        (* Warnung Revisionsschalter Aus *)
        ayWarningReporter[2].proPrio := 1;
	    ayWarningReporter[2].proHandLokal :=    xVerdiRevisionSwitchOff; 
        ayWarningReporter[2].metReport(			xSetReportIn					:= xVerdiRevisionSwitchOff,
												iReportID						:= 2,
												enReportTypeIn					:= CtaAppReport.enReportType.Warning,  
												enReportAcknowledgeTypeIn   	:= CtaAppReport.enReportAcknowledgeType.Auto,
												tDelay							:= T#0S, 
												ITF_BMK_IN						:= THIS^,			              
												pstReportTextListIn				:= ADR(GlobalKonstant.stReportTextListWarning),
												stOptionalReportText		    := '',   
												iRetryTilReportLock 		    := 0, 
												xResetCount         		    := FALSE,  
												tReset						    := T#24H);     

        (* Warnung Hand Aus *)      
        ayWarningReporter[3].proPrio := 3;  
		ayWarningReporter[3].proHandLokal :=    xIsHandOff; 
        ayWarningReporter[3].metReport(			xSetReportIn					:= xIsHandOff,
												iReportID						:= 3,
												enReportTypeIn					:= CtaAppReport.enReportType.Warning,  
												enReportAcknowledgeTypeIn   	:= CtaAppReport.enReportAcknowledgeType.Auto,
												tDelay							:= T#0S, 
												ITF_BMK_IN						:= THIS^,			              
												pstReportTextListIn				:= ADR(GlobalKonstant.stReportTextListWarning),
												stOptionalReportText		    := '',   
												iRetryTilReportLock 		    := 0, 
												xResetCount         		    := FALSE,  
												tReset						    := T#24H);                                  
                                
        (* Warnung Hand Ein *)    
        ayWarningReporter[4].proPrio := 3; 
		ayWarningReporter[4].proHandLokal :=    xIsHandOn;
        ayWarningReporter[4].metReport(			xSetReportIn					:= xIsHandOn,
												iReportID						:= 4,
												enReportTypeIn					:= CtaAppReport.enReportType.Warning,  
												enReportAcknowledgeTypeIn   	:= CtaAppReport.enReportAcknowledgeType.Auto,
												tDelay							:= T#0S, 
												ITF_BMK_IN						:= THIS^,			              
												pstReportTextListIn				:= ADR(GlobalKonstant.stReportTextListWarning),
												stOptionalReportText		    := '',   
												iRetryTilReportLock 		    := 0, 
												xResetCount         		    := FALSE,  
												tReset						    := T#24H);   
 
        (* Warnung Handmodul Motor *)   
        ayWarningReporter[5].proPrio := 4;  
		ayWarningReporter[5].proHandLokal :=    xVerdichterHand;
        ayWarningReporter[5].metReport(			xSetReportIn					:= xVerdichterHand,
												iReportID						:= 5,
												enReportTypeIn					:= CtaAppReport.enReportType.Warning,  
												enReportAcknowledgeTypeIn   	:= CtaAppReport.enReportAcknowledgeType.Auto,
												tDelay							:= T#0S, 
												ITF_BMK_IN						:= THIS^,			              
												pstReportTextListIn				:= ADR(GlobalKonstant.stReportTextListWarning),
												stOptionalReportText		    := '',   
												iRetryTilReportLock 		    := 0, 
												xResetCount         		    := FALSE,  
												tReset						    := T#24H);                                                   
(* Sync Reports *)                                         
FOR difor := LOWER_BOUND(ayErrorReporter,1) TO UPPER_BOUND(ayErrorReporter,1) DO
	fbReportManager.metSyncReporter(ayErrorReporter[difor]);	
END_FOR;
FOR difor := LOWER_BOUND(ayWarningReporter,1) TO UPPER_BOUND(ayWarningReporter,1) DO
	fbReportManager.metSyncReporter(ayWarningReporter[difor]);	
END_FOR;
                                                                             
_xIsError   := scEWI.iError <> 0;
_xIsWarning := scEWI.iWarning <> 0;
END_ACTION

PROPERTY proCountedError : INT
GET
proCountedError := fbReportManager.proAnzError;
END_GET
END_PROPERTY

PROPERTY proCountedInfo : INT
GET
proCountedInfo := fbReportManager.proAnzInfo;
END_GET
END_PROPERTY

PROPERTY proCountedWarning : INT
GET
proCountedWarning := fbReportManager.proAnzWarning;
END_GET
END_PROPERTY

PROPERTY proITF_REPORTMANAGER : CtaAppReport.ITF_REPORTMANAGER
GET
proITF_REPORTMANAGER := fbReportManager;
END_GET
END_PROPERTY

{attribute 'monitoring' := 'variable'}
PROPERTY proLockDown : BOOL
GET
proLockDown := proIsError;
END_GET
END_PROPERTY

{attribute 'monitoring' := 'variable'}
PROPERTY proAvailable : BOOL
GET
proAvailable := proIsReady;
END_GET
END_PROPERTY

{attribute 'monitoring' := 'variable'}
PROPERTY proAcknowledge : BOOL
GET
proAcknowledge := proIsOn;
END_GET
END_PROPERTY

PROPERTY proITF_EINSATZGRENZE : CtaAppEinsatzDiagramm.ITF_EINSATZGRENZE
SET
ITF_EINSATZGRENZE := proITF_EINSATZGRENZE;
END_SET
GET
proITF_EINSATZGRENZE := ITF_EINSATZGRENZE;
END_GET
END_PROPERTY

PROPERTY proITF_FU : CtaSysFU.ITF_FU_BASE
SET
ITF_FU_BASE := proITF_FU;
END_SET
GET
proITF_FU := ITF_FU_BASE;
END_GET
END_PROPERTY

ACTION actFU:
IF __QUERYINTERFACE(ITF_FU_BASE,ITF_FU_BASE) THEN
	IF scParameter.scBase.fbxEnableFU.proValue THEN
		ITF_FU_BASE.proEnable	:= TRUE;
		(* Motor Ready *)
		IF scParameter.scInVerdichterReady.fbxInputMb.proValue THEN
			xInVerdichterIsReadyMb               := ITF_FU_BASE.proReady;
		ELSE
			xInVerdichterIsReadyMb               := FALSE;
		END_IF;
		(* Motor is ON *)
		IF scParameter.scInVerdichterOn.fbxInputMb.proValue THEN
			xInVerdichterIsOnMb                  := ITF_FU_BASE.proAcknowledge;
		ELSE
			xInVerdichterIsOnMb                  := FALSE;
		END_IF;
		(* Motor no error *)
		IF scParameter.scInVerdichterNoError.fbxInputMb.proValue THEN
			xInVerdichterNoErrorMb               := NOT ITF_FU_BASE.proError;
		ELSE
			xInVerdichterNoErrorMb               := FALSE;
		END_IF;
		(* Revision Switch *)
		IF scParameter.scInVerdiRevisionSwitch.fbxInputMb.proValue THEN
			xInVerdiRevisionSwitchOnMb      := TRUE;				// Platzhalter
		ELSE
			xInVerdiRevisionSwitchOnMb      := FALSE;    
		END_IF;
		(* Fuse Ok *)
		IF scParameter.scFuse.fbxInputMb.proValue THEN    
			xInFuseOkMb                     := TRUE;				// Platzhalter
		ELSE
			xInFuseOkMb                     := FALSE;
		END_IF;
		(* Motor Protection *)
		IF scParameter.scVerdichterFuse.fbxInputMb.proValue THEN
			xInVerdichterFuseOkMb                := TRUE;			// Platzhalter
		ELSE
			xInVerdichterFuseOkMb                := FALSE;
		END_IF;
		(* Motor Hand *)
		IF scParameter.scInVerdichterHand.fbxInputMb.proValue THEN
			xInVerdichterHandMb                  := ITF_FU_BASE.proHandLokal;
		ELSE
			xInVerdichterHandMb                  := FALSE;
		END_IF; 
		(*Actual Value*)
		IF scParameter.scInVerdichterActualValue.fbxInputMb.proValue THEN
			rInActualValue					:= ITF_FU_BASE.proAcknowledge_Hz;
		ELSE
			rInActualValue					:= 0;
		END_IF
		(* Release *)
		IF scParameter.scFU.fbxReleaseMb.proValue THEN
			ITF_FU_BASE.proRelease := xOn;
		ELSE
			ITF_FU_BASE.proRelease := FALSE;
		END_IF;
		(* Sollwert *)
		IF scParameter.scFU.fbxSollWertMb.proValue THEN
			ITF_FU_BASE.proRelease_Hz := rOnHz;
		ELSE
			ITF_FU_BASE.proRelease_Hz := 0;
		END_IF;		
	ELSE
		ITF_FU_BASE.proRelease := FALSE;
		IF NOT ITF_FU_BASE.proAcknowledge THEN
			ITF_FU_BASE.proEnable	:= FALSE;
		END_IF
	END_IF;	
	ITF_FU_BASE.proITF_ReportManager := fbReportManager;	
ELSE   
    xInVerdichterIsReadyMb              := FALSE;
    xInVerdichterIsOnMb                 := FALSE;
    xInVerdichterNoErrorMb              := FALSE;
    xInVerdiRevisionSwitchOnMb      	:= FALSE; 
    xInFuseOkMb                     	:= FALSE;
    xInVerdichterFuseOkMb               := FALSE;
    xInVerdichterHandMb                 := FALSE;
END_IF;
END_ACTION

PROPERTY proITF_LEISTUNGVENTILE : CtaSysLeistungventile.ITF_LEISTUNGSVENTILE_BASE
SET
ITF_LEISTUNGSVENTILE := proITF_LEISTUNGVENTILE;
END_SET
GET
proITF_LEISTUNGVENTILE := ITF_LEISTUNGSVENTILE;
END_GET
END_PROPERTY

ACTION actLeistungsventile:
IF __QUERYINTERFACE(ITF_LEISTUNGSVENTILE,ITF_LEISTUNGSVENTILE) THEN
	ITF_LEISTUNGSVENTILE.proRelease := xRelease;
END_IF
END_ACTION

END_FUNCTION_BLOCK

// 21 Interface/ITF_VERDICHTER
INTERFACE ITF_VERDICHTER EXTENDS CtaAppBmk.ITF_BMK, CtaAppModbusSpezifikation.ITF_MODBUS_SPEZIFIKATION

{attribute 'hide'} 
PROPERTY INTERNAL proModbusTest : BOOL
GET
END_GET
SET
END_SET
END_PROPERTY

{warning disable C0410}
PROPERTY proModbusStateWord : REFERENCE TO ARRAY[0..3] OF WORD
{warning restore C0410}
GET
END_GET
END_PROPERTY

PROPERTY P_scFU_fbxReleaseMb : CtaSysConfig.ITF_DATATYPE
GET
END_GET
END_PROPERTY

PROPERTY P_scFU_fbxSollWertMb : CtaSysConfig.ITF_DATATYPE
GET
END_GET
END_PROPERTY

{attribute 'hide'} 
PROPERTY proConfigError : BOOL
GET
END_GET
END_PROPERTY

PROPERTY proAtIconNr : UINT
SET
END_SET
GET
END_GET
END_PROPERTY

PROPERTY P_scBase_fbxEnable : CtaSysConfig.ITF_DATATYPE
GET
END_GET
END_PROPERTY

PROPERTY P_scBase_fbxRegulatet : CtaSysConfig.ITF_DATATYPE
GET
END_GET
END_PROPERTY

PROPERTY P_scBase_fbxEnableFU : CtaSysConfig.ITF_DATATYPE
GET
END_GET
END_PROPERTY

PROPERTY P_scBase_fbrYMax : CtaSysConfig.ITF_DATATYPE
GET
END_GET
END_PROPERTY

PROPERTY P_scBase_fbrYMin : CtaSysConfig.ITF_DATATYPE
GET
END_GET
END_PROPERTY

PROPERTY P_scBase_fbtDelayOnToOn : CtaSysConfig.ITF_DATATYPE
GET
END_GET
END_PROPERTY

PROPERTY P_scBase_fbtDelayOffToOn : CtaSysConfig.ITF_DATATYPE
GET
END_GET
END_PROPERTY

PROPERTY P_scData_fbudiOperatingHours : CtaSysConfig.ITF_DATATYPE
GET
END_GET
END_PROPERTY

PROPERTY P_scData_fbudiOperationStarts : CtaSysConfig.ITF_DATATYPE
GET
END_GET
END_PROPERTY

PROPERTY P_scFuse_fbxDoesAlarm : CtaSysConfig.ITF_DATATYPE
GET
END_GET
END_PROPERTY

PROPERTY P_scFuse_fbxEnable : CtaSysConfig.ITF_DATATYPE
GET
END_GET
END_PROPERTY

PROPERTY P_scFuse_fbxInputMb : CtaSysConfig.ITF_DATATYPE
GET
END_GET
END_PROPERTY

PROPERTY P_scInfluxDb_fbxEnable : CtaSysConfig.ITF_DATATYPE
GET
END_GET
END_PROPERTY

PROPERTY P_scIO_RevisionSwitch_fbxEnable : CtaSysConfig.ITF_DATATYPE
GET
END_GET
END_PROPERTY

PROPERTY P_scIO_RevisionSwitch_fbxInputMb : CtaSysConfig.ITF_DATATYPE
GET
END_GET
END_PROPERTY

PROPERTY P_scIO_IsReady_fbxEnable : CtaSysConfig.ITF_DATATYPE
GET
END_GET
END_PROPERTY

PROPERTY P_scIO_IsReady_fbxInputMb : CtaSysConfig.ITF_DATATYPE
GET
END_GET
END_PROPERTY

PROPERTY P_scIO_IsHand_fbxEnable : CtaSysConfig.ITF_DATATYPE
GET
END_GET
END_PROPERTY

PROPERTY P_scIO_IsHand_fbxInputMb : CtaSysConfig.ITF_DATATYPE
GET
END_GET
END_PROPERTY

PROPERTY P_scIO_IsOn_fbxInputMb : CtaSysConfig.ITF_DATATYPE
GET
END_GET
END_PROPERTY

PROPERTY P_scIO_IsOn_fbxEnable : CtaSysConfig.ITF_DATATYPE
GET
END_GET
END_PROPERTY

PROPERTY P_scIO_IsOn_fbtDelayStart : CtaSysConfig.ITF_DATATYPE
GET
END_GET
END_PROPERTY

PROPERTY P_scIO_IsOn_fbxDoesAlarm : CtaSysConfig.ITF_DATATYPE
GET
END_GET
END_PROPERTY

PROPERTY P_scIO_IsOn_fbtDelayRun : CtaSysConfig.ITF_DATATYPE
GET
END_GET
END_PROPERTY

PROPERTY P_scIO_IsOn_fbiTypeOfAck : CtaSysConfig.ITF_DATATYPE
GET
END_GET
END_PROPERTY

PROPERTY P_scIO_IsOn_fbiMaxErrorRetryAllowed : CtaSysConfig.ITF_DATATYPE
GET
END_GET
END_PROPERTY

PROPERTY P_scIO_IsNoError_fbxEnable : CtaSysConfig.ITF_DATATYPE
GET
END_GET
END_PROPERTY

PROPERTY P_scIO_IsNoError_fbxInputMb : CtaSysConfig.ITF_DATATYPE
GET
END_GET
END_PROPERTY

PROPERTY P_scIO_IsNoError_fbxDoesAlarm : CtaSysConfig.ITF_DATATYPE
GET
END_GET
END_PROPERTY

PROPERTY P_scIO_IsNoError_fbtDelayStartSps : CtaSysConfig.ITF_DATATYPE
GET
END_GET
END_PROPERTY

PROPERTY P_scIO_IsNoError_fbtDelayRun : CtaSysConfig.ITF_DATATYPE
GET
END_GET
END_PROPERTY

PROPERTY P_scIO_IsNoError_fbiTypeOfAck : CtaSysConfig.ITF_DATATYPE
GET
END_GET
END_PROPERTY

PROPERTY P_scIO_IsNoError_fbiMaxErrorRetryAllowed : CtaSysConfig.ITF_DATATYPE
GET
END_GET
END_PROPERTY

PROPERTY P_scIO_IsValue_fbxInputMb : CtaSysConfig.ITF_DATATYPE
GET
END_GET
END_PROPERTY

PROPERTY P_scIO_IsValue_fbxEnable : CtaSysConfig.ITF_DATATYPE
GET
END_GET
END_PROPERTY

PROPERTY P_scIO_IsValue_fbxDoesAlarm : CtaSysConfig.ITF_DATATYPE
GET
END_GET
END_PROPERTY

PROPERTY P_scIO_IsValue_fbtDelayStart : CtaSysConfig.ITF_DATATYPE
GET
END_GET
END_PROPERTY

PROPERTY P_scIO_IsValue_fbtDelayRun : CtaSysConfig.ITF_DATATYPE
GET
END_GET
END_PROPERTY

PROPERTY P_scIO_IsValue_fbiTypeOfAck : CtaSysConfig.ITF_DATATYPE
GET
END_GET
END_PROPERTY

PROPERTY P_scIO_IsValue_fbiMaxErrorRetryAllowed : CtaSysConfig.ITF_DATATYPE
GET
END_GET
END_PROPERTY

PROPERTY P_scIO_IsValue_fbrMaxDiff : CtaSysConfig.ITF_DATATYPE
GET
END_GET
END_PROPERTY

PROPERTY P_scManual_fbrManualOnY : CtaSysConfig.ITF_DATATYPE
GET
END_GET
END_PROPERTY

PROPERTY P_scManual_fbuiManualState : CtaSysConfig.ITF_DATATYPE
GET
END_GET
END_PROPERTY

PROPERTY P_scManual_fbxAlowManualOn : CtaSysConfig.ITF_DATATYPE
GET
END_GET
END_PROPERTY

PROPERTY P_scVerdichterFuse_fbxDoesAlarm : CtaSysConfig.ITF_DATATYPE
GET
END_GET
END_PROPERTY

PROPERTY P_scVerdichterFuse_fbxEnable : CtaSysConfig.ITF_DATATYPE
GET
END_GET
END_PROPERTY

PROPERTY P_scVerdichterFuse_fbxInputMb : CtaSysConfig.ITF_DATATYPE
GET
END_GET
END_PROPERTY

PROPERTY proRefToRonYDumper : REFERENCE TO CtaAppDumper.fbDumper
GET
END_GET
END_PROPERTY

{attribute 'hide'} 
PROPERTY INTERNAL proCountedError : INT
GET
END_GET
END_PROPERTY

{attribute 'hide'} 
PROPERTY INTERNAL proCountedInfo : INT
GET
END_GET
END_PROPERTY

{attribute 'hide'} 
PROPERTY INTERNAL proITF_REPORTMANAGER : CtaAppReport.ITF_REPORTMANAGER
GET
END_GET
END_PROPERTY

{attribute 'hide'} 
PROPERTY INTERNAL proCountedWarning : INT
GET
END_GET
END_PROPERTY

PROPERTY proCountedHours : UDINT
GET
END_GET
END_PROPERTY

PROPERTY proCountedStarts : UDINT
GET
END_GET
END_PROPERTY

PROPERTY INTERNAL proGetDI_VerdichterHand : BOOL
GET
END_GET
END_PROPERTY

{attribute 'hide'} 
PROPERTY proNotShowDI_VerdichterHand : BOOL
GET
END_GET
END_PROPERTY

PROPERTY proHandModul_ITF : CtaSysIO.ITF_IO
GET
END_GET
END_PROPERTY

PROPERTY proGetAI_ActualValue : REAL
GET
END_GET
END_PROPERTY

PROPERTY proNotShowAI_ActualValue : BOOL
GET
END_GET
END_PROPERTY

PROPERTY proActualValue_ITF : CtaSysIO.ITF_IO
GET
END_GET
END_PROPERTY

{attribute 'hide'} 
PROPERTY proNotShowDI_NoError : BOOL
GET
END_GET
END_PROPERTY

PROPERTY INTERNAL proGetDI_NoError : BOOL
GET
END_GET
END_PROPERTY

PROPERTY proNoError_ITF : CtaSysIO.ITF_IO
GET
END_GET
END_PROPERTY

{attribute 'hide'} 
PROPERTY proNotShowDI_RevisionSwitchOk : BOOL
GET
END_GET
END_PROPERTY

PROPERTY INTERNAL proGetDI_RevisionSwitchOK : BOOL
GET
END_GET
END_PROPERTY

PROPERTY proRevisionSwitch_ITF : CtaSysIO.ITF_IO
GET
END_GET
END_PROPERTY

{attribute 'hide'} 
PROPERTY proNotShowDI_IsOn : BOOL
GET
END_GET
END_PROPERTY

PROPERTY INTERNAL proGetDI_IsOn : BOOL
GET
END_GET
END_PROPERTY

PROPERTY proIsOn_ITF : CtaSysIO.ITF_IO
GET
END_GET
END_PROPERTY

{attribute 'hide'} 
PROPERTY proNotShowDI_VerdichterFuseOk : BOOL
GET
END_GET
END_PROPERTY

PROPERTY INTERNAL proGetDI_VerdichterFuseOk : BOOL
GET
END_GET
END_PROPERTY

PROPERTY proVerdichterFuse_ITF : CtaSysIO.ITF_IO
GET
END_GET
END_PROPERTY

{attribute 'hide'} 
PROPERTY proNotShowDI_FuseOk : BOOL
GET
END_GET
END_PROPERTY

PROPERTY INTERNAL proGetDI_FuseOK : BOOL
GET
END_GET
END_PROPERTY

PROPERTY proFuse_ITF : CtaSysIO.ITF_IO
GET
END_GET
END_PROPERTY

{attribute 'hide'} 
PROPERTY proNotShowDI_Ready : BOOL
GET
END_GET
END_PROPERTY

PROPERTY INTERNAL proGetDI_IsReady : BOOL
GET
END_GET
END_PROPERTY

PROPERTY proReady_ITF : CtaSysIO.ITF_IO
GET
END_GET
END_PROPERTY

PROPERTY proOn_ITF : CtaSysIO.ITF_IO
GET
END_GET
END_PROPERTY

PROPERTY proOnY_ITF : CtaSysIO.ITF_IO
GET
END_GET
END_PROPERTY

PROPERTY proLeistung : REAL
GET
END_GET
END_PROPERTY

PROPERTY proIsOn : BOOL
GET
END_GET
END_PROPERTY

PROPERTY proIsOnY : REAL
GET
END_GET
END_PROPERTY

{attribute 'hide'} 
PROPERTY INTERNAL proEnSymbol : STRING
GET
END_GET
END_PROPERTY

{attribute 'hide'} 
PROPERTY INTERNAL proStateSymbol : STRING
GET
END_GET
END_PROPERTY

PROPERTY proIsRegulatet : BOOL
GET
END_GET
END_PROPERTY

PROPERTY proIsHandOnOrOff : BOOL
GET
END_GET
END_PROPERTY

PROPERTY proRestartLockTime : TIME
GET
END_GET
END_PROPERTY

PROPERTY proOn : BOOL
GET
END_GET
END_PROPERTY

PROPERTY proCommutingProtectionTime : TIME
GET
END_GET
END_PROPERTY

PROPERTY proCommutingProtectionAktive : BOOL
GET
END_GET
END_PROPERTY

PROPERTY proRestartLockAktive : BOOL
GET
END_GET
END_PROPERTY

PROPERTY proIsReady : BOOL
GET
END_GET
END_PROPERTY

PROPERTY proAuto : BOOL
GET
END_GET
SET
END_SET
END_PROPERTY

PROPERTY proHandOn : BOOL
SET
END_SET
GET
END_GET
END_PROPERTY

PROPERTY proIsError : BOOL
GET
END_GET
END_PROPERTY

PROPERTY proIsWarning : BOOL
GET
END_GET
END_PROPERTY

PROPERTY proEn : BOOL
GET
END_GET
SET
END_SET
END_PROPERTY

PROPERTY proOnY : REAL
GET
END_GET
END_PROPERTY

PROPERTY proHardWareHandModulAktive : BOOL
GET
END_GET
END_PROPERTY

PROPERTY proIsEnabled : BOOL
GET
END_GET
END_PROPERTY

PROPERTY proMotorIsOn : BOOL
GET
END_GET
END_PROPERTY

PROPERTY proHandOff : BOOL
SET
END_SET
GET
END_GET
END_PROPERTY

PROPERTY proRevisionSwitchOk : BOOL
GET
END_GET
END_PROPERTY

PROPERTY proHandOnY : REAL
SET
END_SET
GET
END_GET
END_PROPERTY

PROPERTY proOnHz : REAL
GET
END_GET
END_PROPERTY

PROPERTY proResetVerdiTime : BOOL
SET
END_SET
GET
END_GET
END_PROPERTY

{attribute 'monitoring' := 'variable'}
PROPERTY proLockDown : BOOL
GET
END_GET
END_PROPERTY

{attribute 'monitoring' := 'variable'}
PROPERTY proAvailable : BOOL
GET
END_GET
END_PROPERTY

{attribute 'monitoring' := 'variable'}
PROPERTY proAcknowledge : BOOL
GET
END_GET
END_PROPERTY

PROPERTY proITF_EINSATZGRENZE : CtaAppEinsatzDiagramm.ITF_EINSATZGRENZE
SET
END_SET
GET
END_GET
END_PROPERTY

PROPERTY proITF_FU : CtaSysFU.ITF_FU_BASE
SET
END_SET
GET
END_GET
END_PROPERTY

PROPERTY proITF_LEISTUNGVENTILE : CtaSysLeistungventile.ITF_LEISTUNGSVENTILE_BASE
SET
END_SET
GET
END_GET
END_PROPERTY

END_INTERFACE

// 30 Program Organization Units/fcGetBigerStringValue
FUNCTION fcGetBigerStringValue : INT
VAR_INPUT
    st1     :   STRING(255);
    st2     :   STRING(255);
END_VAR
VAR
    diFor: DINT;
    diMax: DINT;
END_VAR

IF LEN(st1) > LEN(st2) THEN
    diMax := LEN(st2); 
    fcGetBigerStringValue := 1;
ELSIF LEN(st1) < LEN(st2) THEN
    diMax := LEN(st1);
    fcGetBigerStringValue := 2;     
ELSE
    diMax := LEN(st1);    
END_IF;
FOR diFor := 0 TO  diMax DO
    IF st1[diFor] > st2[diFor] THEN
        fcGetBigerStringValue := 1;  
        EXIT; 
    ELSIF st1[diFor] < st2[diFor] THEN
        fcGetBigerStringValue := 2;  
        EXIT;
    END_IF;
END_FOR;

END_FUNCTION

// 30 Program Organization Units/fcCheckQuerryAndIconReturn
FUNCTION fcCheckQuerryAndIconReturn : BOOL
VAR_INPUT
	_ITF_IN			: 	ITF_VERDICHTER;
	_uiIconNr_IN	:	UINT;
END_VAR

IF __QUERYINTERFACE(_ITF_IN,_ITF_IN) THEN
	fcCheckQuerryAndIconReturn := TRUE;	
	_ITF_IN.proAtIconNr := _uiIconNr_IN;
ELSE
	fcCheckQuerryAndIconReturn :=  FALSE;
END_IF

END_FUNCTION

// 40 Visualizations/POPUP/POPUP_VERDICHTER
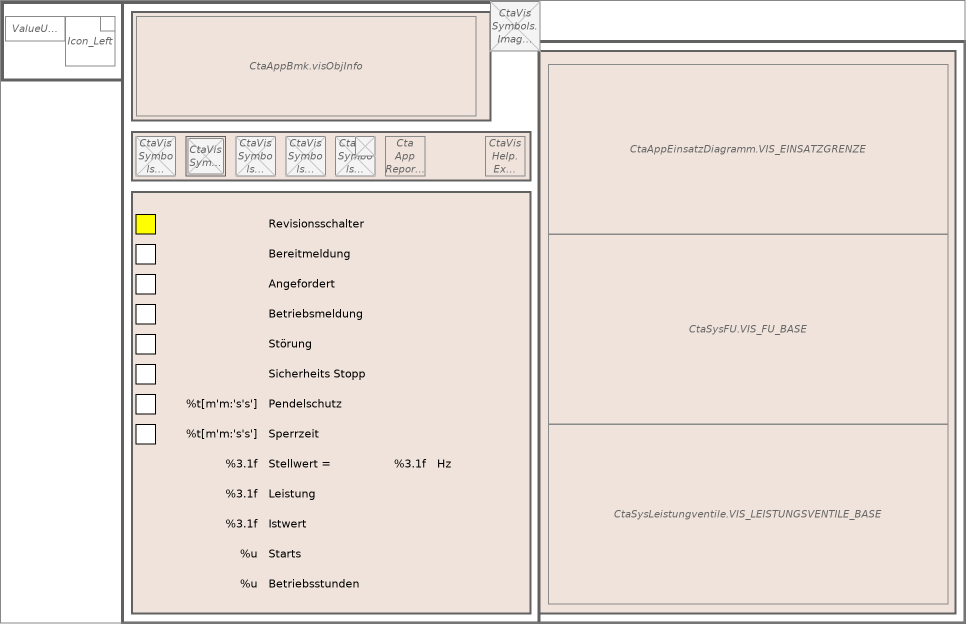
VISUALIZATION POPUP_VERDICHTER  // 966x624
VAR_INPUT
    ITF_VERDICHTERIN    :   ITF_VERDICHTER;
	stExklParameter		:	STRING[40];	
	uiPopUpGruppe 		:	UINT;
END_VAR
    RoundedRectangle (517,40 449x584)
    RoundedRectangle (527,50 429x564)
    RoundedRectangle (1,1 160x80)
    RoundedRectangle (121,1 419x623)
    RoundedRectangle (131,11 360x110)
    RoundedRectangle (131,191 400x423)
    RoundedRectangle (131,131 400x50)
    Frame (136,16 340x100)
        shows CtaAppBmk.visObjInfo(ITF_BMK_IN := ITF_VERDICHTERIN)
    Image (490,1 50x50), image: CtaVisSymbols.ImagePool.close_solo_black
        OnMouseClick:  Dialog=Current Dialog, Result=None, NumpadKeypadSet=True
    Frame (131,204 399x400), frame switch variable: uiPopUpGruppe
        shows VIS_VERDICHTER_OVERVIEW(ITF_VERDICHTERIN := ITF_VERDICHTERIN)
        shows VIS_VERDICHTER_MANUAL(ITF_VERDICHTERIN := ITF_VERDICHTERIN)
        shows VIS_VERDICHTER_PARAMETER(ITF_VERDICHTERIN := ITF_VERDICHTERIN)
        shows VIS_VERDICHTER_IO(ITF_VERDICHTERIN := ITF_VERDICHTERIN)
        shows VERDICHTER_BUS(ITF_VERDICHTERIN := ITF_VERDICHTERIN)
        shows VIS_VERDICHTER_REPORTS(ITF_VERDICHTERIN := ITF_VERDICHTERIN)
    Frame (131,136 399x40)
        shows VIS_VERDICHTER_LISTE(uiPopUpGruppe := uiPopUpGruppe, xHand := ITF_VERDICHTERIN.proIsHandOnOrOff, xHandOff := ITF_VERDICHTERIN.proHandOff, ITF_REPORTMANAGER_IN := ITF_VERDICHTERIN.proITF_REPORTMANAGER, xBusTestAktiv := ITF_VERDICHTERIN.proModbusTest, stExklParameter_IN := stExklParameter)
        pReferences[0]: AnzError=ITF_VERDICHTERIN.proCountedError, AnzWarning=ITF_VERDICHTERIN.proCountedWarning
    Frame (5,16 110x50), input disabled if: TRUE, frame switch variable: ITF_VERDICHTERIN.proAtIconNr
        shows VIS_VERDICHTER_LEFT_ABOVE(ITF_VERDICHTER_IN := ITF_VERDICHTERIN, stExklParameter := stExklParameter)
        shows VIS_VERDICHTER_LEFT_BELOW(ITF_VERDICHTER_IN := ITF_VERDICHTERIN, stExklParameter := stExklParameter)
        shows VIS_VERDICHTER_RIGHT_ABOVE(ITF_VERDICHTER_IN := ITF_VERDICHTERIN, stExklParameter := stExklParameter)
        shows VIS_VERDICHTER_RIGHT_BELOW(ITF_VERDICHTER_IN := ITF_VERDICHTERIN, stExklParameter := stExklParameter)
    Frame (548,64 400x170)
        shows CtaAppEinsatzDiagramm.VIS_EINSATZGRENZE(ITF_EINSATZGRENZEIn := ITF_VERDICHTERIN.proITF_EINSATZGRENZE)
    Frame (548,234 400x190)
        shows CtaSysFU.VIS_FU_BASE(ITF_FU_BASEIn := ITF_VERDICHTERIN.proITF_FU)
    Frame (548,424 400x180)
        shows CtaSysLeistungventile.VIS_LEISTUNGSVENTILE_BASE(ITF_LEISTUNGSVENTILE_BASEIn := ITF_VERDICHTERIN.proITF_LEISTUNGVENTILE)
    InvisibleInput (131,3 360x48)
END_VISUALIZATION

// 40 Visualizations/POPUP/VIS_VERDICHTER_LISTE
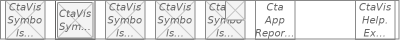
VISUALIZATION VIS_VERDICHTER_LISTE  // 400x40
VAR_IN_OUT
	uiPopUpGruppe 			:	UINT;
END_VAR
VAR_INPUT
    xHand           		: 	BOOL;
    xHandOff        		: 	BOOL;
    ITF_REPORTMANAGER_IN 	: 	CtaAppReport.ITF_REPORTMANAGER;
    xBusTestAktiv   		: 	BOOL;	
	stExklParameter_IN		:	STRING[40];
END_VAR
    Group (5,0 40x40)
        RoundedRectangle (0,0 40x40), colour toggle: uiPopUpGruppe = 0
            OnMouseDown: execute { uiPopUpGruppe := 0; }
        Image (0,0 40x40), image: CtaVisSymbols.ImagePool.eye
            OnMouseDown: execute { uiPopUpGruppe := 0; }
    Group (105,0 40x40)
        RoundedRectangle (0,0 40x40), colour toggle: uiPopUpGruppe = 2
            OnMouseDown: execute { uiPopUpGruppe := 2; }
        Image (0,0 40x40), image: CtaVisSymbols.ImagePool.gear
            OnMouseDown: execute { uiPopUpGruppe := 2; }
    Group (55,0 40x40)
        RoundedRectangle (0,0 40x40), colour toggle: uiPopUpGruppe = 1
            OnMouseDown: execute { uiPopUpGruppe := 1; }
        Image (2,2 36x36), image: CtaVisSymbols.ImagePool.front_hand_Black
            OnMouseDown: execute { uiPopUpGruppe := 1; }
        Image (2,2 36x36), invisible if: NOT xHand, image: CtaVisSymbols.ImagePool.front_hand_Yellow
            OnMouseDown: execute { uiPopUpGruppe := 1; }
        Image (2,2 36x36), invisible if: NOT xHandOff, image: CtaVisSymbols.ImagePool.front_hand_Yellow_Off
            OnMouseDown: execute { uiPopUpGruppe := 1; }
    Group (155,0 40x40)
        RoundedRectangle (0,0 40x40), colour toggle: uiPopUpGruppe = 3
            OnMouseDown: execute { uiPopUpGruppe := 3; }
        Image (0,0 40x40), image: CtaVisSymbols.ImagePool.dip-switch
            OnMouseDown: execute { uiPopUpGruppe := 3; }
    Group (205,0 40x40)
        RoundedRectangle (0,0 40x40), colour toggle: uiPopUpGruppe = 4
            OnMouseDown: execute { uiPopUpGruppe := 4; }
        Image (0,0 40x40), image: CtaVisSymbols.ImagePool.lan
            OnMouseDown: execute { uiPopUpGruppe := 4; }
        Image (20,0 20x20), invisible if: NOT xBusTestAktiv, image: CtaVisSymbols.ImagePool.front_hand_Yellow
            OnMouseDown: execute { uiPopUpGruppe := 4; }
    Group (255,0 40x40)
        RoundedRectangle (0,0 40x40), colour toggle: uiPopUpGruppe = 5
            OnMouseDown: execute { uiPopUpGruppe := 5; }
        Frame (0,0 40x40), input disabled if: TRUE
            shows CtaAppReport.VIS_ANZ_REPORTS_MODUL(ITF_REPORTMANAGER_IN := ITF_REPORTMANAGER_IN)
            OnMouseDown: execute { uiPopUpGruppe := 5; }
    Group (355,0 40x40)
        RoundedRectangle (0,0 40x40), invisible if: stExklParameter_IN = ' '
        Frame (0,0 40x40)
            shows CtaVisHelp.ExkParameterSymbol(stExklParameter := stExklParameter_IN)
END_VISUALIZATION

// 40 Visualizations/ICON/VERDICHTER_RIGHT/VERDICHTER_RIGHT_ABOVE/VIS_VERDICHTER_RigthAboveCheckQuerry
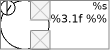
VISUALIZATION VIS_VERDICHTER_RigthAboveCheckQuerry  // 110x50
VAR_INPUT
    ITF_VERDICHTER_IN   :   ITF_VERDICHTER;	
    stExklParameter		:   STRING[40];	
END_VAR
    Frame (0,0 110x50)
        shows VIS_VERDICHTER_RigthAboveCheckIsEnabled(ITF_VERDICHTER_IN := ITF_VERDICHTER_IN, stExklParameter := stExklParameter)
END_VISUALIZATION

// 40 Visualizations/ICON/VERDICHTER_RIGHT/VERDICHTER_RIGHT_ABOVE/VIS_VERDICHTER_RIGHT_ABOVE
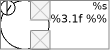
VISUALIZATION VIS_VERDICHTER_RIGHT_ABOVE  // 110x50
VAR_INPUT
    ITF_VERDICHTER_IN   :   ITF_VERDICHTER;	
END_VAR
VAR_INPUT CONSTANT
    stExklParameter		:   STRING[40] := '';	
END_VAR
VAR CONSTANT
	uiIconNr		: UINT := 2;
END_VAR
    Frame (0,0 110x50), invisible if: NOT fcCheckQuerryAndIconReturn(_ITF_IN := ITF_VERDICHTER_IN, _uiIconNr_IN := uiIconNr)
        shows VIS_VERDICHTER_RigthAboveCheckQuerry(ITF_VERDICHTER_IN := ITF_VERDICHTER_IN, stExklParameter := stExklParameter)
END_VISUALIZATION

// 40 Visualizations/ICON/VERDICHTER_RIGHT/VERDICHTER_RIGHT_ABOVE/VIS_VERDICHTER_RigthAboveCheckIsEnabled
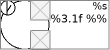
VISUALIZATION VIS_VERDICHTER_RigthAboveCheckIsEnabled  // 110x50
VAR_INPUT
    ITF_VERDICHTER_IN   :   ITF_VERDICHTER;
    stExklParameter		:   STRING[40];	
END_VAR
    Frame (0,0 50x50), invisible if: NOT ITF_VERDICHTER_IN.proIsEnabled
        shows Icon_Right(ITF_VERDICHTER_IN := ITF_VERDICHTER_IN)
        shows Value_Right()
    Frame (50,0 60x25), invisible if: NOT ITF_VERDICHTER_IN.proIsEnabled
        shows ValueUpDwn(ITF_VERDICHTER_IN := ITF_VERDICHTER_IN, uiTextAusrichtung := 4)
    Frame (0,0 15x15), invisible if: NOT ITF_VERDICHTER_IN.proIsEnabled
        shows CommandOn(ITF_VERDICHTER_IN := ITF_VERDICHTER_IN)
    Rectangle (0,0 110x50)
        OnMouseClick:  Dialog=POPUP_VERDICHTER, Parameters={stExklParameter: stExklParameter, ITF_VERDICHTERIN: ITF_VERDICHTER_IN, uiPopUpGruppe: 0}, OpenCentered=True
END_VISUALIZATION

// 40 Visualizations/ICON/VERDICHTER_BASE/CommandOn
VISUALIZATION CommandOn  // 15x15
VAR_INPUT
    ITF_VERDICHTER_IN   :   ITF_VERDICHTER;	
END_VAR
    Ellipse (0,0 15x15), colour toggle: ITF_VERDICHTER_IN.proOn
    Line (7,15) (7,10)
    Line (7,5) (7,0)
    Line (7,11) (11,5), invisible if: ITF_VERDICHTER_IN.proOn
    Line (7,15) (7,0), invisible if: NOT ITF_VERDICHTER_IN.proOn
END_VISUALIZATION

// 40 Visualizations/ICON/VERDICHTER_BASE/ICON/Icon_Left
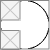
VISUALIZATION Icon_Left  // 50x50
VAR_INPUT
    ITF_VERDICHTER_IN   :   ITF_VERDICHTER;	
END_VAR
    Ellipse (0,0 49x49), colour toggle: ITF_VERDICHTER_IN.proMotorIsOn, invisible if: ITF_VERDICHTER_IN.proIsError
    Ellipse (0,0 49x49), colour toggle: ITF_VERDICHTER_IN.proIsError
    Image (0,0 20x20), invisible if: NOT ITF_VERDICHTER_IN.proIsWarning, image: CtaVisSymbols.ImagePool.CtaWarning
    Image (0,30 20x20), invisible if: NOT ITF_VERDICHTER_IN.proIsHandOnOrOff, image: CtaVisSymbols.ImagePool.front_hand_Yellow
    Image (0,30 20x20), invisible if: NOT ITF_VERDICHTER_IN.proHandOff, image: CtaVisSymbols.ImagePool.front_hand_Yellow_Off
END_VISUALIZATION

// 40 Visualizations/POPUP/PARAMETER/VIS_VERDICHTER_PARAMETER
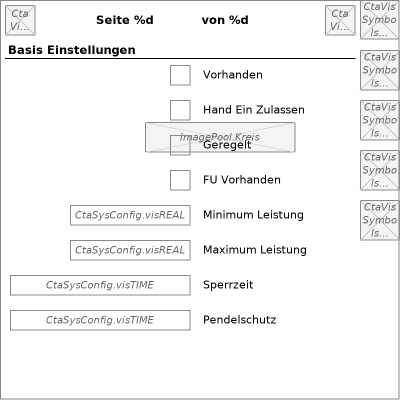
VISUALIZATION VIS_VERDICHTER_PARAMETER  // 400x400
VAR_INPUT
    ITF_VERDICHTERIN : ITF_VERDICHTER;
END_VAR
VAR
    uiParameterGruppe : UINT;
END_VAR
    Image (145,122 150x30), image: ImagePool.Kreis
    Frame (360,0 40x300)
        shows VIS_VERDICHTER_PARAMETER_LISTE(uiParameterGruppe := uiParameterGruppe)
    Frame (0,0 360x400), frame switch variable: uiParameterGruppe
        shows VIS_VERDICHTER_PARAMETER_BASE(ITF_VERDICHTERIN := ITF_VERDICHTERIN)
        shows VIS_VERDICHTER_PARAMETER_FUSES(ITF_VERDICHTERIN := ITF_VERDICHTERIN)
        shows VIS_VERDICHTER_PARAMETER_IO(ITF_VERDICHTERIN := ITF_VERDICHTERIN)
        shows VIS_VERDICHTER_PARAMETER_DATA(ITF_VERDICHTERIN := ITF_VERDICHTERIN)
        shows VIS_VERDICHTER_PARAMETER_TRENDLOG(ITF_VERDICHTERIN := ITF_VERDICHTERIN)
        pReferences[0]: ITF_Parameter=ITF_Parameter
        pReferences[1]: ITF_Parameter=ITF_Parameter
        pReferences[3]: ITF_Parameter=ITF_Parameter
END_VISUALIZATION

// 40 Visualizations/POPUP/PARAMETER/VIS_VERDICHTER_PARAMETER_LISTE
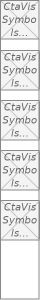
VISUALIZATION VIS_VERDICHTER_PARAMETER_LISTE  // 40x300
VAR_IN_OUT
	uiParameterGruppe : UINT;
END_VAR
    RoundedRectangle (0,150 39x39), colour toggle: uiParameterGruppe = 3
        OnMouseDown: execute { uiParameterGruppe := 3; }
    RoundedRectangle (0,100 39x39), colour toggle: uiParameterGruppe = 2
        OnMouseDown: execute { uiParameterGruppe := 2; }
    RoundedRectangle (0,50 39x39), colour toggle: uiParameterGruppe = 1
        OnMouseDown: execute { uiParameterGruppe := 1; }
    RoundedRectangle (0,0 39x39), colour toggle: uiParameterGruppe = 0
        OnMouseDown: execute { uiParameterGruppe := 0; }
    RoundedRectangle (0,200 39x39), colour toggle: uiParameterGruppe = 4
        OnMouseDown: execute { uiParameterGruppe := 4; }
    Image (0,0 39x39), image: CtaVisSymbols.ImagePool.engine
        OnMouseDown: execute { uiParameterGruppe := 0; }
    Image (0,50 40x40), image: CtaVisSymbols.ImagePool.electric_bolt_24dp_000000_FILL0_wght400_GRAD0_opsz24
        OnMouseDown: execute { uiParameterGruppe := 1; }
    Image (0,100 40x40), image: CtaVisSymbols.ImagePool.dip-switch
        OnMouseDown: execute { uiParameterGruppe := 2; }
    Image (0,150 40x40), image: CtaVisSymbols.ImagePool.database_black
        OnMouseDown: execute { uiParameterGruppe := 3; }
    Image (0,200 40x40), image: CtaVisSymbols.ImagePool.sine-wave
        OnMouseDown: execute { uiParameterGruppe := 4; }
END_VISUALIZATION

// 40 Visualizations/POPUP/MANUAL/VIS_VERDICHTER_MANUAL
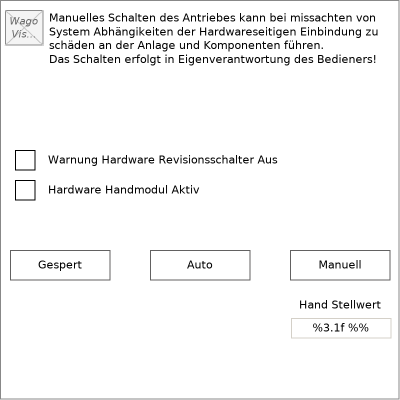
VISUALIZATION VIS_VERDICHTER_MANUAL  // 400x400
VAR_INPUT
    ITF_VERDICHTERIN    :   ITF_VERDICHTER;	
END_VAR
    Label (46,10 350x100), "Manuelles Schalten des Antriebes kann bei missachten von System Abhängikeiten der Hardwareseitigen Einbindung zu schäden an der Anlage und Komponenten führen. Das Schalten erfolgt in Eigenverantwortung des Bedieners!"
    Textfield (291,318 100x20), "%3.1f %%", text variable: ITF_VERDICHTERIN.proHandOnY, invisible if: NOT ITF_VERDICHTERIN.proIsRegulatet
        OnMouseClick: write the text variable via InputWithLimits, min 0, max 100, title 'Stellwert'
    Image (5,10 38x35), image: WagoVisuIcons.WagoIcons.2
    Label (290,295 100x20), "Hand Stellwert"
    Rectangle (15,180 20x20), colour toggle: ITF_VERDICHTERIN.proHardWareHandModulAktive, invisible if: NOT ITF_VERDICHTERIN.proHardWareHandModulAktive
    Label (45,180 200x20), "Hardware Handmodul Aktiv", invisible if: NOT ITF_VERDICHTERIN.proHardWareHandModulAktive
    Label (45,150 350x20), "Warnung Hardware Revisionsschalter Aus", invisible if: ITF_VERDICHTERIN.proRevisionSwitchOk
    Rectangle (15,150 20x20), colour toggle: NOT ITF_VERDICHTERIN.proRevisionSwitchOk, invisible if: ITF_VERDICHTERIN.proRevisionSwitchOk
    RoundedRectangle (10,250 100x30), "Gespert", colour toggle: ITF_VERDICHTERIN.proHandOff
        toggle ITF_VERDICHTERIN.proHandOff
    RoundedRectangle (150,250 100x30), "Auto", colour toggle: ITF_VERDICHTERIN.proAuto
        toggle ITF_VERDICHTERIN.proAuto
    RoundedRectangle (290,250 100x30), "Manuell", colour toggle: ITF_VERDICHTERIN.proHandOn
        toggle ITF_VERDICHTERIN.proHandOn
END_VISUALIZATION

// 40 Visualizations/POPUP/OVERVIEW/VIS_VERDICHTER_OVERVIEW
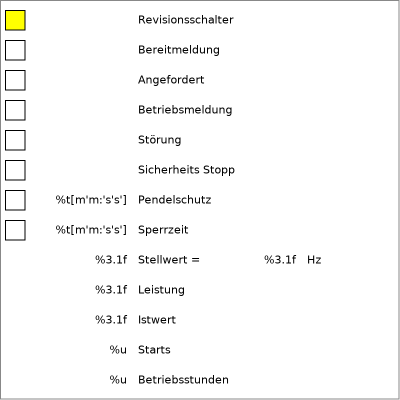
VISUALIZATION VIS_VERDICHTER_OVERVIEW  // 400x400
VAR_INPUT
    ITF_VERDICHTERIN    :   ITF_VERDICHTER;	
END_VAR
    Label (135,370 200x20), "Betriebsstunden"
    Textfield (30,370 100x20), "%u", text variable: ITF_VERDICHTERIN.proCountedHours
    Label (135,340 200x20), "Starts"
    Textfield (30,340 100x20), "%u", text variable: ITF_VERDICHTERIN.proCountedStarts
    Label (135,310 200x20), "Istwert", invisible if: NOT ITF_VERDICHTERIN.proIsRegulatet
    Textfield (30,310 100x20), "%3.1f", text variable: ITF_VERDICHTERIN.proIsOnY, invisible if: NOT ITF_VERDICHTERIN.proIsRegulatet
    Label (135,280 200x20), "Leistung", invisible if: NOT ITF_VERDICHTERIN.proIsRegulatet
    Textfield (30,280 100x20), "%3.1f", text variable: ITF_VERDICHTERIN.proLeistung, invisible if: NOT ITF_VERDICHTERIN.proIsRegulatet
    Label (304,250 48x20), "Hz", invisible if: NOT ITF_VERDICHTERIN.proIsRegulatet
    Textfield (199,250 100x20), "%3.1f", text variable: ITF_VERDICHTERIN.proOnHz, invisible if: NOT ITF_VERDICHTERIN.proIsRegulatet
    Label (135,250 200x20), "Stellwert =", invisible if: NOT ITF_VERDICHTERIN.proIsRegulatet
    Textfield (30,250 100x20), "%3.1f", text variable: ITF_VERDICHTERIN.proOnY, invisible if: NOT ITF_VERDICHTERIN.proIsRegulatet
    Rectangle (0,186 400x59)
        OnMouseClick:  Dialog=ResetVerdiTime, Parameters={ITF_VERDICHTER_IN: ITF_VERDICHTERIN}, Selected={0: }, OpenCentered=True
    Label (135,220 200x20), "Sperrzeit"
    Textfield (30,220 100x20), "%t[m'm:'s's']", text variable: ITF_VERDICHTERIN.proRestartLockTime
    Rectangle (5,220 20x20), colour toggle: ITF_VERDICHTERIN.proRestartLockAktive
    Label (135,190 200x20), "Pendelschutz"
    Textfield (30,190 100x20), "%t[m'm:'s's']", text variable: ITF_VERDICHTERIN.proCommutingProtectionTime
    Rectangle (5,190 20x20), colour toggle: ITF_VERDICHTERIN.proCommutingProtectionAktive
    Label (135,160 200x20), "Sicherheits Stopp"
    Rectangle (5,160 20x20)
    Label (135,130 200x20), "Störung"
    Rectangle (5,130 20x20), colour toggle: ITF_VERDICHTERIN.proIsError
    Label (135,100 200x20), "Betriebsmeldung"
    Rectangle (5,100 20x20), colour toggle: ITF_VERDICHTERIN.proMotorIsOn
    Label (135,70 200x20), "Angefordert"
    Rectangle (5,70 20x20), colour toggle: ITF_VERDICHTERIN.proOn
    Label (135,40 200x20), "Bereitmeldung"
    Rectangle (5,40 20x20), colour toggle: ITF_VERDICHTERIN.proIsReady
    Label (135,10 200x20), "Revisionsschalter"
    Rectangle (5,10 20x20), colour toggle: ITF_VERDICHTERIN.proRevisionSwitchOk
END_VISUALIZATION

// 40 Visualizations/POPUP/BUS/VERDICHTER_BUS
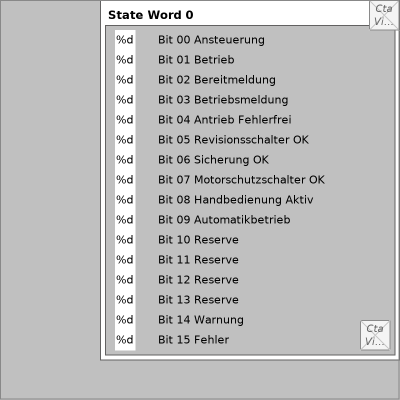
VISUALIZATION VERDICHTER_BUS  // 400x400
VAR_INPUT
    ITF_VERDICHTERIN    :   ITF_VERDICHTER;	
END_VAR
    Frame (100,0 300x360)
        shows VERDICHTER_BUS_CS(ITF_VERDICHTERIn := ITF_VERDICHTERIN, ayStateWord := ITF_VERDICHTERIN.proModbusStateWord)
        pReferences[0]: ayControllWord=ITF_VERDICHTERIN.proModbusControllWord
END_VISUALIZATION

// 40 Visualizations/POPUP/BUS/VERDICHTER_BUS_SW0_Detail
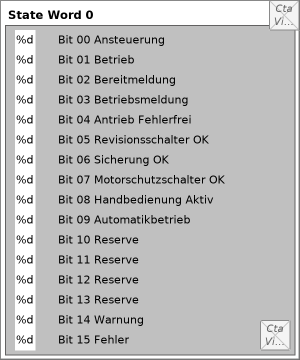
VISUALIZATION VERDICHTER_BUS_SW0_Detail  // 300x360
VAR_IN_OUT
    wDetail     :   WORD;
END_VAR
VAR_INPUT	
    ITF_VERDICHTERIN    :   ITF_VERDICHTER;
END_VAR
VAR_IN_OUT
    xShow       :   BOOL;
END_VAR
    RoundedRectangle (0,0 300x360)
    RoundedRectangle (5,25 290x330)
    Textfield (15,30 20x20), "%d", text variable: TO_WORD(wDetail.0), input disabled if: NOT ITF_VERDICHTERIn.proModbusTest
        OnMouseClick: execute { wDetail.0 := NOT wDetail.0; }
    Label (55,30 220x20), "Bit 00 Ansteuerung"
    Textfield (15,50 20x20), "%d", text variable: TO_WORD(wDetail.1), input disabled if: NOT ITF_VERDICHTERIn.proModbusTest
        OnMouseClick: execute { wDetail.1 := NOT wDetail.1; }
    Label (55,50 220x20), "Bit 01 Betrieb"
    Textfield (15,70 20x20), "%d", text variable: TO_WORD(wDetail.2), input disabled if: NOT ITF_VERDICHTERIn.proModbusTest
        OnMouseClick: execute { wDetail.2 := NOT wDetail.2; }
    Label (55,70 220x20), "Bit 02 Bereitmeldung"
    Textfield (15,90 20x20), "%d", text variable: TO_WORD(wDetail.3), input disabled if: NOT ITF_VERDICHTERIn.proModbusTest
        OnMouseClick: execute { wDetail.3 := NOT wDetail.3; }
    Label (55,90 220x20), "Bit 03 Betriebsmeldung"
    Textfield (15,110 20x20), "%d", text variable: TO_WORD(wDetail.4), input disabled if: NOT ITF_VERDICHTERIn.proModbusTest
        OnMouseClick: execute { wDetail.4 := NOT wDetail.4; }
    Label (55,110 220x20), "Bit 04 Antrieb Fehlerfrei"
    Textfield (15,130 20x20), "%d", text variable: TO_WORD(wDetail.5), input disabled if: NOT ITF_VERDICHTERIn.proModbusTest
        OnMouseClick: execute { wDetail.5 := NOT wDetail.5; }
    Label (55,130 220x20), "Bit 05 Revisionsschalter OK"
    Textfield (15,150 20x20), "%d", text variable: TO_WORD(wDetail.6), input disabled if: NOT ITF_VERDICHTERIn.proModbusTest
        OnMouseClick: execute { wDetail.6 := NOT wDetail.6; }
    Label (55,150 220x20), "Bit 06 Sicherung OK"
    Textfield (15,170 20x20), "%d", text variable: TO_WORD(wDetail.7), input disabled if: NOT ITF_VERDICHTERIn.proModbusTest
        OnMouseClick: execute { wDetail.7 := NOT wDetail.7; }
    Label (55,170 220x20), "Bit 07 Motorschutzschalter OK"
    Textfield (15,190 20x20), "%d", text variable: TO_WORD(wDetail.8), input disabled if: NOT ITF_VERDICHTERIn.proModbusTest
        OnMouseClick: execute { wDetail.8 := NOT wDetail.8; }
    Label (55,190 220x20), "Bit 08 Handbedienung Aktiv"
    Textfield (15,210 20x20), "%d", text variable: TO_WORD(wDetail.9), input disabled if: NOT ITF_VERDICHTERIn.proModbusTest
        OnMouseClick: execute { wDetail.9 := NOT wDetail.9; }
    Label (55,210 220x20), "Bit 09 Automatikbetrieb"
    Textfield (15,230 20x20), "%d", text variable: TO_WORD(wDetail.10), input disabled if: NOT ITF_VERDICHTERIn.proModbusTest
        OnMouseClick: execute { wDetail.10 := NOT wDetail.10; }
    Label (55,230 220x20), "Bit 10 Reserve"
    Textfield (15,250 20x20), "%d", text variable: TO_WORD(wDetail.11), input disabled if: NOT ITF_VERDICHTERIn.proModbusTest
        OnMouseClick: execute { wDetail.11 := NOT wDetail.11; }
    Label (55,250 220x20), "Bit 11 Reserve"
    Textfield (15,270 20x20), "%d", text variable: TO_WORD(wDetail.12), input disabled if: NOT ITF_VERDICHTERIn.proModbusTest
        OnMouseClick: execute { wDetail.12 := NOT wDetail.12; }
    Label (55,270 220x20), "Bit 12 Reserve"
    Textfield (15,290 20x20), "%d", text variable: TO_WORD(wDetail.13), input disabled if: NOT ITF_VERDICHTERIn.proModbusTest
        OnMouseClick: execute { wDetail.13 := NOT wDetail.13; }
    Label (55,290 220x20), "Bit 13 Reserve"
    Textfield (15,310 20x20), "%d", text variable: TO_WORD(wDetail.14), input disabled if: NOT ITF_VERDICHTERIn.proModbusTest
        OnMouseClick: execute { wDetail.14 := NOT wDetail.14; }
    Label (55,310 220x20), "Bit 14 Warnung"
    Textfield (15,330 20x20), "%d", text variable: TO_WORD(wDetail.15), input disabled if: NOT ITF_VERDICHTERIn.proModbusTest
        OnMouseClick: execute { wDetail.15 := NOT wDetail.15; }
    Label (55,330 220x20), "Bit 15 Fehler"
    Image (269,0 30x30), image: CtaVisSymbols.ImagePool.close_solo_black
        OnMouseClick: execute { xShow := FALSE; ITF_vERDICHTERIN.proModbusTest := FALSE; }
    Label (5,0 150x30), "State Word 0"
    Image (260,320 30x30), invisible if: ITF_VERDICHTERIN.proModbusTest, image: CtaVisSymbols.ImagePool.front_hand_Black
        OnMouseClick: execute { ITF_VERDICHTERIN.proModbusTest := TRUE; }
    Image (260,320 30x30), invisible if: NOT ITF_VERDICHTERIN.proModbusTest, image: CtaVisSymbols.ImagePool.front_hand_Yellow
        OnMouseClick: execute { ITF_VERDICHTERIN.proModbusTest := False; }
END_VISUALIZATION

// 40 Visualizations/POPUP/BUS/VERDICHTER_BUS_CS
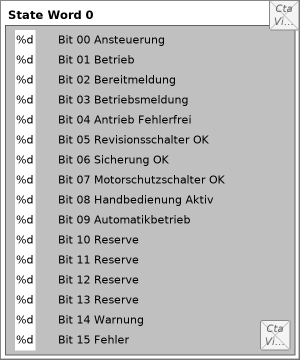
VISUALIZATION VERDICHTER_BUS_CS  // 300x360
VAR_INPUT
    ITF_VERDICHTERIn        :   ITF_VERDICHTER;
    ayStateWord     :   REFERENCE TO ARRAY[0..3] OF WORD;
END_VAR
VAR
    xShowCw :   BOOL;
    xShowSw :   BOOL;
    xShowSw1:   BOOL;
    xShowSw2:   BOOL;
	xShowSw3:   BOOL;
END_VAR
    Label (140,290 120x20), "State Word 3"
    Textfield (0,170 130x20), "%b", text variable: ayStateWord[0]
        OnMouseDown: write the text variable via Default
    Label (140,170 120x20), "State Word 0"
    Label (140,210 120x20), "State Word 1"
    Textfield (0,210 130x20), "%d", text variable: ayStateWord[1]
    Label (140,250 120x20), "State Word 2"
    Textfield (0,250 130x20), "%d", text variable: ayStateWord[2]
    Textfield (0,290 130x20), "%d", text variable: ayStateWord[3]
    Image (265,165 30x30), image: CtaVisSymbols.ImagePool.information-variant
        OnMouseClick: execute {
            xShowCw := FALSE;
            xShowSw := TRUE;
            xShowSw1:= FALSE;
            xShowSw2:= FALSE;
            xShowSw3:= FALSE;
        }
    Image (265,205 30x30), image: CtaVisSymbols.ImagePool.information-variant
        OnMouseClick: execute {
            xShowCw := FALSE;
            xShowSw := FALSE;
            xShowSw1:= TRUE;
            xShowSw2:= FALSE;
            xShowSw3:= FALSE;
        }
    Image (265,245 30x30), image: CtaVisSymbols.ImagePool.information-variant
        OnMouseClick: execute {
            xShowCw := FALSE;
            xShowSw := FALSE;
            xShowSw1:= FALSE;
            xShowSw2:= TRUE;
            xShowSw3:= FALSE;
        }
    Image (265,285 30x30), image: CtaVisSymbols.ImagePool.information-variant
        OnMouseClick: execute {
            xShowCw := FALSE;
            xShowSw := FALSE;
            xShowSw1:= FALSE;
            xShowSw2:= FALSE;
            xShowSw3:= TRUE;
        }
    Frame (0,0 300x360), invisible if: NOT xShowSw3
        shows VERDICHTER_BUS_SW3_Detail(wDetail := ayStateWord[3], ITF_VERDICHTERIN := ITF_VERDICHTERIn, xShow := xShowSw3)
        p731600746: ayStateWord[3]
        p2277378067: ITF_VERDICHTERIn
        p499328597: xShowSw3
    Frame (0,0 300x360), invisible if: NOT xShowSw2
        shows VERDICHTER_BUS_SW2_Detail(wDetail := ayStateWord[2], ITF_VERDICHTERIN := ITF_VERDICHTERIn, xShow := xShowSw2)
    Frame (0,0 300x360), invisible if: NOT xShowSw1
        shows VERDICHTER_BUS_SW1_Detail(wDetail := ayStateWord[1], ITF_VERDICHTERIN := ITF_VERDICHTERIn, xShow := xShowSw1)
    Frame (0,0 300x360), invisible if: NOT xShowSw
        shows VERDICHTER_BUS_SW0_Detail(wDetail := ayStateWord[0], ITF_VERDICHTERIN := ITF_VERDICHTERIn, xShow := xShowSw)
END_VISUALIZATION

// 40 Visualizations/POPUP/BUS/VERDICHTER_BUS_SW1_Detail
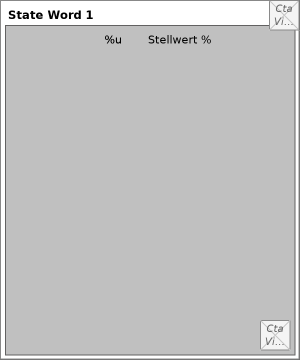
VISUALIZATION VERDICHTER_BUS_SW1_Detail  // 300x360
VAR_IN_OUT
    wDetail     :   WORD;
END_VAR
VAR_INPUT	
    ITF_VERDICHTERIN    :   ITF_VERDICHTER;
END_VAR
VAR_IN_OUT
    xShow       :   BOOL;
END_VAR
    RoundedRectangle (0,0 300x360)
    RoundedRectangle (5,25 290x330)
    Image (269,0 30x30), image: CtaVisSymbols.ImagePool.close_solo_black
        OnMouseClick: execute { xShow := FALSE; ITF_VERDICHTERIN.proModbusTest := FALSE; }
    Label (5,0 150x30), "State Word 1"
    Label (145,30 120x20), "Stellwert %"
    Textfield (15,30 110x20), "%u", text variable: wDetail, input disabled if: NOT ITF_VERDICHTERIn.proModbusTest
        OnMouseClick: write the text variable via InputWithLimits, min 0, max 100
    Textfield (15,30 110x20), "%u", text variable: wDetail, invisible if: ITF_VERDICHTERIN.proModbusTest
    Image (260,320 30x30), invisible if: ITF_VERDICHTERIN.proModbusTest, image: CtaVisSymbols.ImagePool.front_hand_Black
        OnMouseClick: execute { ITF_VERDICHTERIN.proModbusTest := TRUE; }
    Image (260,320 30x30), invisible if: NOT ITF_VERDICHTERIN.proModbusTest, image: CtaVisSymbols.ImagePool.front_hand_Yellow
        OnMouseClick: execute { ITF_VERDICHTERIN.proModbusTest := False; }
END_VISUALIZATION

// 40 Visualizations/POPUP/BUS/VERDICHTER_BUS_SW2_Detail
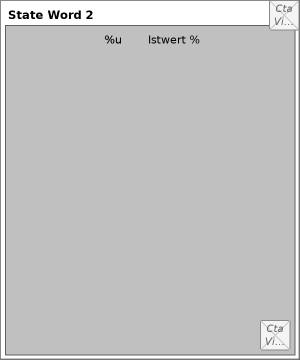
VISUALIZATION VERDICHTER_BUS_SW2_Detail  // 300x360
VAR_IN_OUT
    wDetail             :   WORD;
END_VAR
VAR_INPUT	
    ITF_VERDICHTERIN       :   ITF_VERDICHTER;
END_VAR
VAR_IN_OUT
    xShow               :   BOOL;
END_VAR
    RoundedRectangle (0,0 300x360)
    RoundedRectangle (5,25 290x330)
    Image (269,0 30x30), image: CtaVisSymbols.ImagePool.close_solo_black
        OnMouseClick: execute { xShow := FALSE; ITF_VERDICHTERIN.proModbusTest := FALSE; }
    Label (5,0 150x30), "State Word 2"
    Label (145,30 120x20), "Istwert %"
    Textfield (15,30 110x20), "%u", text variable: wDetail, input disabled if: NOT ITF_VERDICHTERIn.proModbusTest
        OnMouseClick: write the text variable via InputWithLimits, min 0, max 100
    Textfield (15,30 110x20), "%u", text variable: wDetail, invisible if: ITF_VERDICHTERIN.proModbusTest
    Image (260,320 30x30), invisible if: ITF_VERDICHTERIN.proModbusTest, image: CtaVisSymbols.ImagePool.front_hand_Black
        OnMouseClick: execute { ITF_VERDICHTERIN.proModbusTest := TRUE; }
    Image (260,320 30x30), invisible if: NOT ITF_VERDICHTERIN.proModbusTest, image: CtaVisSymbols.ImagePool.front_hand_Yellow
        OnMouseClick: execute { ITF_VERDICHTERIN.proModbusTest := False; }
END_VISUALIZATION

// 40 Visualizations/POPUP/REPORTS/VIS_VERDICHTER_REPORTS
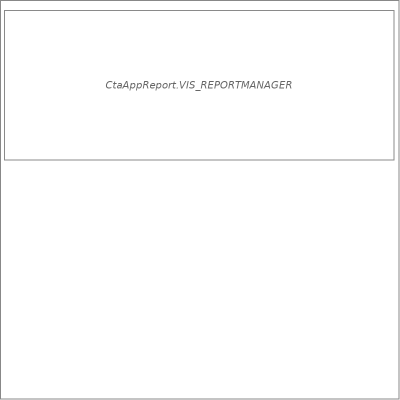
VISUALIZATION VIS_VERDICHTER_REPORTS  // 400x400
VAR_INPUT
    ITF_VERDICHTERIN    :   ITF_VERDICHTER;	
END_VAR
    Frame (4,10 390x150)
        shows CtaAppReport.VIS_REPORTMANAGER(ITF_REPORTMANAGER := ITF_VERDICHTERIN.proITF_REPORTMANAGER)
END_VISUALIZATION

// 40 Visualizations/POPUP/PARAMETER/VERDICHTER_ParameterBase/VIS_VERDICHTER_PARAMETER_BASE0
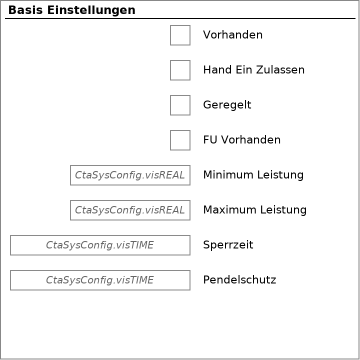
VISUALIZATION VIS_VERDICHTER_PARAMETER_BASE0  // 360x360
VAR_INPUT
    ITF_VERDICHTERIN : ITF_VERDICHTER;
END_VAR
    Frame (170,25 20x20)
        shows CtaSysConfig.visBOOL(visfbBOOLIn := ITF_VERDICHTERIN.P_scBase_fbxEnable)
    Label (200,25 150x20), "Vorhanden"
    Frame (170,95 20x20)
        shows CtaSysConfig.visBOOL(visfbBOOLIn := ITF_VERDICHTERIN.P_scBase_fbxRegulatet)
    Label (200,95 150x20), "Geregelt"
    Frame (170,130 20x20)
        shows CtaSysConfig.visBOOL(visfbBOOLIn := ITF_VERDICHTERIN.P_scBase_fbxEnableFU)
    Label (200,130 150x20), "FU Vorhanden"
    Frame (70,165 120x20)
        shows CtaSysConfig.visREAL(visfbREALIn := ITF_VERDICHTERIN.P_scBase_fbrYMin, stPhysikalischeEinheit := '%')
    Label (200,165 150x20), "Minimum Leistung"
    Frame (70,200 120x20)
        shows CtaSysConfig.visREAL(visfbREALIn := ITF_VERDICHTERIN.P_scBase_fbrYMax, stPhysikalischeEinheit := '%')
    Label (200,200 150x20), "Maximum Leistung"
    Frame (10,235 180x20)
        shows CtaSysConfig.visTIME(visfbTIMEIn := ITF_VERDICHTERIN.P_scBase_fbtDelayOffToOn)
    Label (200,235 150x20), "Sperrzeit"
    Label (200,270 150x20), "Pendelschutz"
    Frame (10,270 180x20)
        shows CtaSysConfig.visTIME(visfbTIMEIn := ITF_VERDICHTERIN.P_scBase_fbtDelayOnToOn)
    Label (5,0 350x20), "Basis Einstellungen"
    Frame (170,60 20x20)
        shows CtaSysConfig.visBOOL(visfbBOOLIn := ITF_VERDICHTERIN.P_scManual_fbxAlowManualOn)
    Label (200,60 150x20), "Hand Ein Zulassen"
    Line (5,18) (355,18)
END_VISUALIZATION

// 40 Visualizations/POPUP/PARAMETER/VERDICHTER_ParameterBase/VIS_VERDICHTER_PARAMETER_BASE
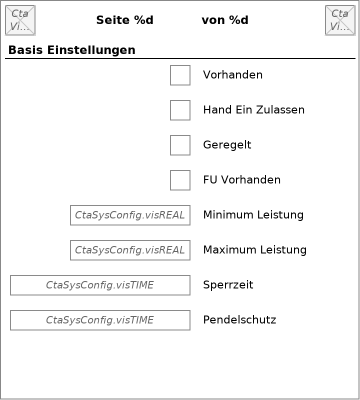
VISUALIZATION VIS_VERDICHTER_PARAMETER_BASE  // 360x400
VAR_INPUT
    ITF_VERDICHTERIN : ITF_VERDICHTER;
END_VAR
VAR
    uiPage  :   UINT;
    uiMin   :   UINT    := 0;
    uiMax   :   UINT    := 0;
END_VAR
    Image (5,5 30x30), invisible if: uiPage = uiMin, image: CtaVisSymbols.ImagePool.arrow-left_square
        OnMouseClick: execute {
            uiPage := uiPage - 1;
            IF uiPage <= uiMin THEN
                uiPage := uiMin;
            END_IF;
        }
    Image (325,5 30x30), invisible if: uiPage = uiMax, image: CtaVisSymbols.ImagePool.arrow-right_square
        OnMouseClick: execute {
            uiPage := uiPage + 1;
            IF uiPage >= uiMax THEN
                uiPage := uiMax;
            END_IF;
        }
    Frame (0,40 360x360), frame switch variable: uiPage
        shows VIS_VERDICHTER_PARAMETER_BASE0(ITF_VERDICHTERIN := ITF_VERDICHTERIN)
        shows VIS_VERDICHTER_PARAMETER_BASE1(ITF_Parameter := ITF_Parameter)
        pReferences[0]: ITF_Parameter=ITF_Parameter
    Textfield (175,5 100x30), "von %d", text variable: uiMax
    Textfield (75,5 100x30), "Seite %d", text variable: uiPage
END_VISUALIZATION

// 40 Visualizations/POPUP/PARAMETER/VERDICHTER_Data/VIS_VERDICHTER_PARAMETER_DATA0
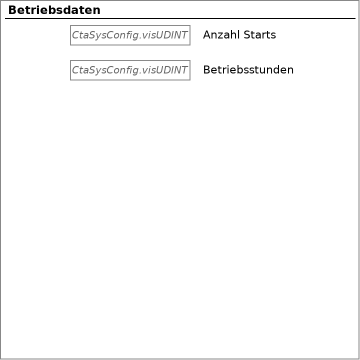
VISUALIZATION VIS_VERDICHTER_PARAMETER_DATA0  // 360x360
VAR_INPUT
    ITF_VERDICHTERIN : ITF_VERDICHTER;
END_VAR
    Label (200,25 150x20), "Anzahl Starts"
    Label (200,60 150x20), "Betriebsstunden"
    Label (5,0 350x20), "Betriebsdaten"
    Frame (70,25 120x20)
        shows CtaSysConfig.visUDINT(visfbUDINTIn := ITF_VERDICHTERIN.P_scData_fbudiOperationStarts)
    Frame (70,60 120x20)
        shows CtaSysConfig.visUDINT(visfbUDINTIn := ITF_VERDICHTERIN.P_scData_fbudiOperatingHours)
    Line (5,18) (355,18)
END_VISUALIZATION

// 40 Visualizations/POPUP/PARAMETER/VERDICHTER_Data/VIS_VERDICHTER_PARAMETER_DATA
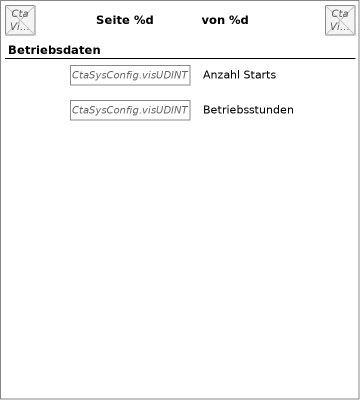
VISUALIZATION VIS_VERDICHTER_PARAMETER_DATA  // 360x400
VAR_INPUT
    ITF_VERDICHTERIN : ITF_VERDICHTER;
END_VAR
VAR
    uiPage  :   UINT;
    uiMin   :   UINT    := 0;
    uiMax   :   UINT    := 0;
END_VAR
    Image (5,5 30x30), invisible if: uiPage = uiMin, image: CtaVisSymbols.ImagePool.arrow-left_square
        OnMouseClick: execute {
            uiPage := uiPage - 1;
            IF uiPage <= uiMin THEN
                uiPage := uiMin;
            END_IF;
        }
    Image (325,5 30x30), invisible if: uiPage = uiMax, image: CtaVisSymbols.ImagePool.arrow-right_square
        OnMouseClick: execute {
            uiPage := uiPage + 1;
            IF uiPage >= uiMax THEN
                uiPage := uiMax;
            END_IF;
        }
    Frame (0,40 360x360), frame switch variable: uiPage
        shows VIS_VERDICHTER_PARAMETER_DATA0(ITF_VERDICHTERIN := ITF_VERDICHTERIN)
        shows AT_ParameterIO1(ITF_Parameter := ITF_Parameter)
        pReferences[0]: ITF_Parameter=ITF_Parameter
    Textfield (75,5 100x30), "Seite %d", text variable: uiPage
    Textfield (175,5 100x30), "von %d", text variable: uiMax
END_VISUALIZATION

// 40 Visualizations/POPUP/PARAMETER/VERDICHTER_Fuse/VIS_VERDICHTER_PARAMETER_FUSES0
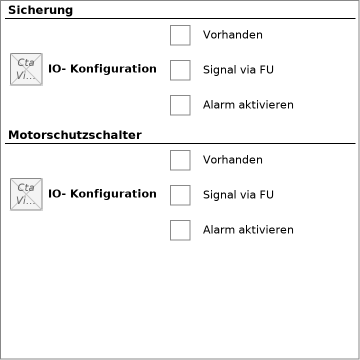
VISUALIZATION VIS_VERDICHTER_PARAMETER_FUSES0  // 360x360
VAR_INPUT
    ITF_VERDICHTERIN  		:	ITF_VERDICHTER;
	ITF_Fuse_IN				:	CtaSysIO.ITF_IO;
	ITF_VerdichterFuse_IN	:	CtaSysIO.ITF_IO;
END_VAR
    Frame (170,25 20x20)
        shows CtaSysConfig.visBOOL(visfbBOOLIn := ITF_VERDICHTERIN.P_scFuse_fbxEnable)
    Label (200,25 150x20), "Vorhanden"
    Frame (170,60 20x20)
        shows CtaSysConfig.visBOOL(visfbBOOLIn := ITF_VERDICHTERIN.P_scFuse_fbxInputMb)
    Label (200,60 150x20), "Signal via FU"
    Frame (170,95 20x20)
        shows CtaSysConfig.visBOOL(visfbBOOLIn := ITF_VERDICHTERIN.P_scFuse_fbxDoesAlarm)
    Label (200,95 150x20), "Alarm aktivieren"
    Label (5,0 350x20), "Sicherung"
    Label (5,125 350x20), "Motorschutzschalter"
    Frame (170,150 20x20)
        shows CtaSysConfig.visBOOL(visfbBOOLIn := ITF_VERDICHTERIN.P_scVerdichterFuse_fbxEnable)
    Label (200,150 150x20), "Vorhanden"
    Frame (170,185 20x20)
        shows CtaSysConfig.visBOOL(visfbBOOLIn := ITF_VERDICHTERIN.P_scVerdichterFuse_fbxInputMb)
    Label (200,185 150x20), "Signal via FU"
    Frame (170,220 20x20)
        shows CtaSysConfig.visBOOL(visfbBOOLIn := ITF_VERDICHTERIN.P_scVerdichterFuse_fbxDoesAlarm)
    Label (200,220 150x20), "Alarm aktivieren"
    Line (5,18) (355,18)
    Line (5,143) (355,143)
    Image (10,53 32x32), invisible if: ITF_Fuse_IN = 0, image: CtaVisSymbols.ImagePool.build
        OnMouseDown:  Dialog=VIS_ANTRIEB_POPUP_IO_ITF, Parameters={ITF_IO_IN: ITF_Fuse_IN}, OpenModal=True, OpenCentered=True
    Image (10,178 32x32), invisible if: ITF_VerdichterFuse_IN = 0, image: CtaVisSymbols.ImagePool.build
        OnMouseDown:  Dialog=VIS_ANTRIEB_POPUP_IO_ITF, Parameters={ITF_IO_IN: ITF_VerdichterFuse_IN}, OpenModal=True, OpenCentered=True
    Label (45,59 120x20), "IO- Konfiguration", invisible if: ITF_Fuse_IN = 0
    Label (45,184 120x20), "IO- Konfiguration", invisible if: ITF_VerdichterFuse_IN = 0
END_VISUALIZATION

// 40 Visualizations/POPUP/PARAMETER/VERDICHTER_Fuse/VIS_VERDICHTER_PARAMETER_FUSES
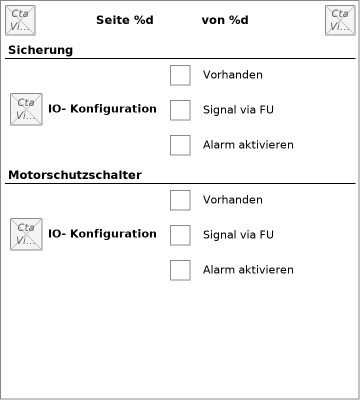
VISUALIZATION VIS_VERDICHTER_PARAMETER_FUSES  // 360x400
VAR_INPUT
    ITF_VERDICHTERIN : ITF_VERDICHTER;
END_VAR
VAR
    uiPage  :   UINT;
    uiMin   :   UINT    := 0;
    uiMax   :   UINT    := 0;
END_VAR
    Image (5,5 30x30), invisible if: uiPage = uiMin, image: CtaVisSymbols.ImagePool.arrow-left_square
        OnMouseClick: execute {
            uiPage := uiPage - 1;
            IF uiPage <= uiMin THEN
                uiPage := uiMin;
            END_IF;
        }
    Image (325,5 30x30), invisible if: uiPage = uiMax, image: CtaVisSymbols.ImagePool.arrow-right_square
        OnMouseClick: execute {
            uiPage := uiPage + 1;
            IF uiPage >= uiMax THEN
                uiPage := uiMax;
            END_IF;
        }
    Frame (0,40 360x360), frame switch variable: uiPage
        shows VIS_VERDICHTER_PARAMETER_FUSES0(ITF_VERDICHTERIN := ITF_VERDICHTERIN, ITF_Fuse_IN := ITF_VERDICHTERIN.proFuse_ITF, ITF_VerdichterFuse_IN := ITF_VERDICHTERIN.proVerdichterFuse_ITF)
        shows AT_ParameterIO1(ITF_Parameter := ITF_Parameter)
        pReferences[0]: ITF_Parameter=ITF_Parameter
    Textfield (75,5 100x30), "Seite %d", text variable: uiPage
    Textfield (175,5 100x30), "von %d", text variable: uiMax
END_VISUALIZATION

// 40 Visualizations/POPUP/PARAMETER/VERDICHTER_IO/VIS_VERDICHTER_PARAMETER_IO0
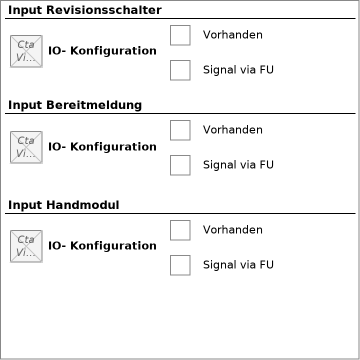
VISUALIZATION VIS_VERDICHTER_PARAMETER_IO0  // 360x360
VAR_INPUT
    ITF_VERDICHTERIN 	: 	ITF_VERDICHTER;
	ITF_RevSwitch_IN	:	CtaSysIO.ITF_IO;
	ITF_VerdiReady_IN	:	CtaSysIO.ITF_IO;
	ITF_VerdiHandMod_IN	:	CtaSysIO.ITF_IO;
END_VAR
    Frame (170,25 20x20)
        shows CtaSysConfig.visBOOL(visfbBOOLIn := ITF_VERDICHTERIN.P_scIO_RevisionSwitch_fbxEnable)
    Label (200,25 150x20), "Vorhanden"
    Frame (170,60 20x20)
        shows CtaSysConfig.visBOOL(visfbBOOLIn := ITF_VERDICHTERIN.P_scIO_RevisionSwitch_fbxInputMb)
    Label (200,60 150x20), "Signal via FU"
    Label (5,0 350x20), "Input Revisionsschalter"
    Label (5,95 350x20), "Input Bereitmeldung"
    Frame (170,120 20x20)
        shows CtaSysConfig.visBOOL(visfbBOOLIn := ITF_VERDICHTERIN.P_scIO_IsReady_fbxEnable)
    Label (200,120 150x20), "Vorhanden"
    Frame (170,155 20x20)
        shows CtaSysConfig.visBOOL(visfbBOOLIn := ITF_VERDICHTERIN.P_scIO_IsReady_fbxInputMb)
    Label (200,155 150x20), "Signal via FU"
    Label (5,195 350x20), "Input Handmodul"
    Frame (170,220 20x20)
        shows CtaSysConfig.visBOOL(visfbBOOLIn := ITF_VERDICHTERIN.P_scIO_IsHand_fbxEnable)
    Label (200,220 150x20), "Vorhanden"
    Frame (170,255 20x20)
        shows CtaSysConfig.visBOOL(visfbBOOLIn := ITF_VERDICHTERIN.P_scIO_IsHand_fbxInputMb)
    Label (200,255 150x20), "Signal via FU"
    Line (5,18) (355,18)
    Line (5,113) (355,113)
    Line (5,213) (355,213)
    Image (10,35 32x32), invisible if: ITF_RevSwitch_IN = 0, input disabled if: ITF_RevSwitch_IN = 0, image: CtaVisSymbols.ImagePool.build
        OnMouseDown:  Dialog=VIS_ANTRIEB_POPUP_IO_ITF, Parameters={ITF_IO_IN: ITF_RevSwitch_IN}, OpenModal=True, OpenCentered=True
    Image (10,131 32x32), invisible if: ITF_VerdiReady_IN = 0, input disabled if: ITF_VerdiReady_IN = 0, image: CtaVisSymbols.ImagePool.build
        OnMouseDown:  Dialog=VIS_ANTRIEB_POPUP_IO_ITF, Parameters={ITF_IO_IN: ITF_VerdiReady_IN}, OpenModal=True, OpenCentered=True
    Image (10,230 32x32), invisible if: ITF_VerdiHandMod_IN = 0, input disabled if: ITF_VerdiHandMod_IN = 0, image: CtaVisSymbols.ImagePool.build
        OnMouseDown:  Dialog=VIS_ANTRIEB_POPUP_IO_ITF, Parameters={ITF_IO_IN: ITF_VerdiHandMod_IN}, OpenModal=True, OpenCentered=True
    Label (45,41 120x20), "IO- Konfiguration", invisible if: ITF_RevSwitch_IN = 0
    Label (45,137 120x20), "IO- Konfiguration", invisible if: ITF_VerdiReady_IN = 0
    Label (45,236 120x20), "IO- Konfiguration", invisible if: ITF_VerdiHandMod_IN = 0
END_VISUALIZATION

// 40 Visualizations/POPUP/PARAMETER/VERDICHTER_IO/VIS_VERDICHTER_PARAMETER_IO1
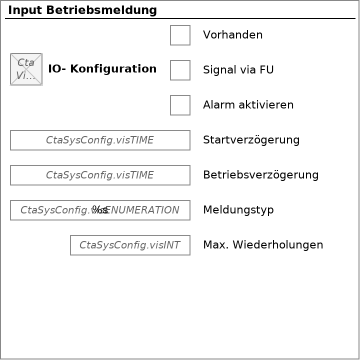
VISUALIZATION VIS_VERDICHTER_PARAMETER_IO1  // 360x360
VAR_INPUT
    ITF_VERDICHTERIN 		:	ITF_VERDICHTER;
	ITF_VerdichterOn_IN		:	CtaSysIO.ITF_IO;	
END_VAR
    Label (5,0 350x20), "Input Betriebsmeldung"
    Frame (170,25 20x20)
        shows CtaSysConfig.visBOOL(visfbBOOLIn := ITF_VERDICHTERIN.P_scIO_IsOn_fbxEnable)
    Label (200,25 150x20), "Vorhanden"
    Frame (170,60 20x20)
        shows CtaSysConfig.visBOOL(visfbBOOLIn := ITF_VERDICHTERIN.P_scIO_IsOn_fbxInputMb)
    Label (200,60 150x20), "Signal via FU"
    Frame (170,95 20x20)
        shows CtaSysConfig.visBOOL(visfbBOOLIn := ITF_VERDICHTERIN.P_scIO_IsOn_fbxDoesAlarm)
    Label (200,95 150x20), "Alarm aktivieren"
    Frame (10,130 180x20)
        shows CtaSysConfig.visTIME(visfbTIMEIn := ITF_VERDICHTERIN.P_scIO_IsOn_fbtDelayStart)
    Label (200,130 150x20), "Startverzögerung"
    Label (200,165 150x20), "Betriebsverzögerung"
    Frame (10,165 180x20)
        shows CtaSysConfig.visTIME(visfbTIMEIn := ITF_VERDICHTERIN.P_scIO_IsOn_fbtDelayRun)
    Label (200,200 150x20), "Meldungstyp"
    Label (200,235 150x20), "Max. Wiederholungen"
    Line (5,18) (355,18)
    Frame (70,235 120x20)
        shows CtaSysConfig.visINT(visfbINTIn := ITF_VERDICHTERIN.P_scIO_IsOn_fbiMaxErrorRetryAllowed)
    Frame (10,200 180x20)
        shows CtaSysConfig.visENUMERATION(visfbENUIn := ITF_VERDICHTERIN.P_scIO_IsOn_fbiTypeOfAck)
    Image (10,53 32x32), invisible if: ITF_VerdichterOn_IN = 0, image: CtaVisSymbols.ImagePool.build
        OnMouseDown:  Dialog=VIS_ANTRIEB_POPUP_IO_ITF, Parameters={ITF_IO_IN: ITF_VerdichterOn_IN}, OpenModal=True, OpenCentered=True
    Label (45,59 120x20), "IO- Konfiguration", invisible if: ITF_VerdichterOn_IN = 0
    Textfield (30,200 140x20), "%s", text list: 'CtaAppReport.txtLibAp99_2enTypeOfAck', text index: CtaSysConfig.fcGetEnumerationId(ITF_VERDICHTERIN.P_scIO_IsOn_fbiTypeOfAck)
END_VISUALIZATION

// 40 Visualizations/POPUP/PARAMETER/VERDICHTER_IO/VIS_VERDICHTER_PARAMETER_IO
